{attribute 'linkalways'} 
{attribute 'no_explicit_call' := 'This FB is a CLASS and must be accessed using methods or properties'}
{attribute 'enable_dynamic_creation'}
FUNCTION_BLOCK UnknownEnumerationError EXTENDS Error
VAR
	enumString : T_MAXSTRING;
END_VAR

PROPERTY PUBLIC ErrorType : T_MAXSTRING
GET
ErrorType := 'UNKNOWN_ENUMERATION_ERROR';
END_GET
END_PROPERTY

METHOD FB_init : BOOL
VAR_INPUT
	bInitRetains : BOOL; // if TRUE, the retain variables are initialized (warm start / cold start)
	bInCopyCode : BOOL;  // if TRUE, the instance afterwards gets moved into the copy code (online change)
	EnumString : T_MAXSTRING;
END_VAR
THIS^.enumString := EnumString;
END_METHOD

PROPERTY PUBLIC Message : T_MAXSTRING
GET
Message := CONCAT('Unknown Enumeration : ', enumString);
END_GET
END_PROPERTY

END_FUNCTION_BLOCK

(* stored: Version 1.1.0.1, ProductVersion 3.1.4024.12
   POU UnknownEnumerationError: Id {19646a27-befd-05cf-2fd3-cc1f5cac95c2}, SpecialFunc None
   Folder Constructor: Id {d8cbdb7d-1052-0ca9-319e-d95fa0e20539}
   Property ErrorType: Id {ad2e303b-e2be-02a5-0600-b83cb2db45b6}
   Get Get: Id {b5e10fe4-943b-0c3b-3591-b3b111608d7f}
   Method FB_init: Id {c8260202-0186-082f-39f1-248a3742d794}
   Property Message: Id {3223dc51-dde2-062b-2d5a-1f5834300a71}
   Get Get: Id {7513b460-bf41-0117-08df-e82e8b461216} *)
